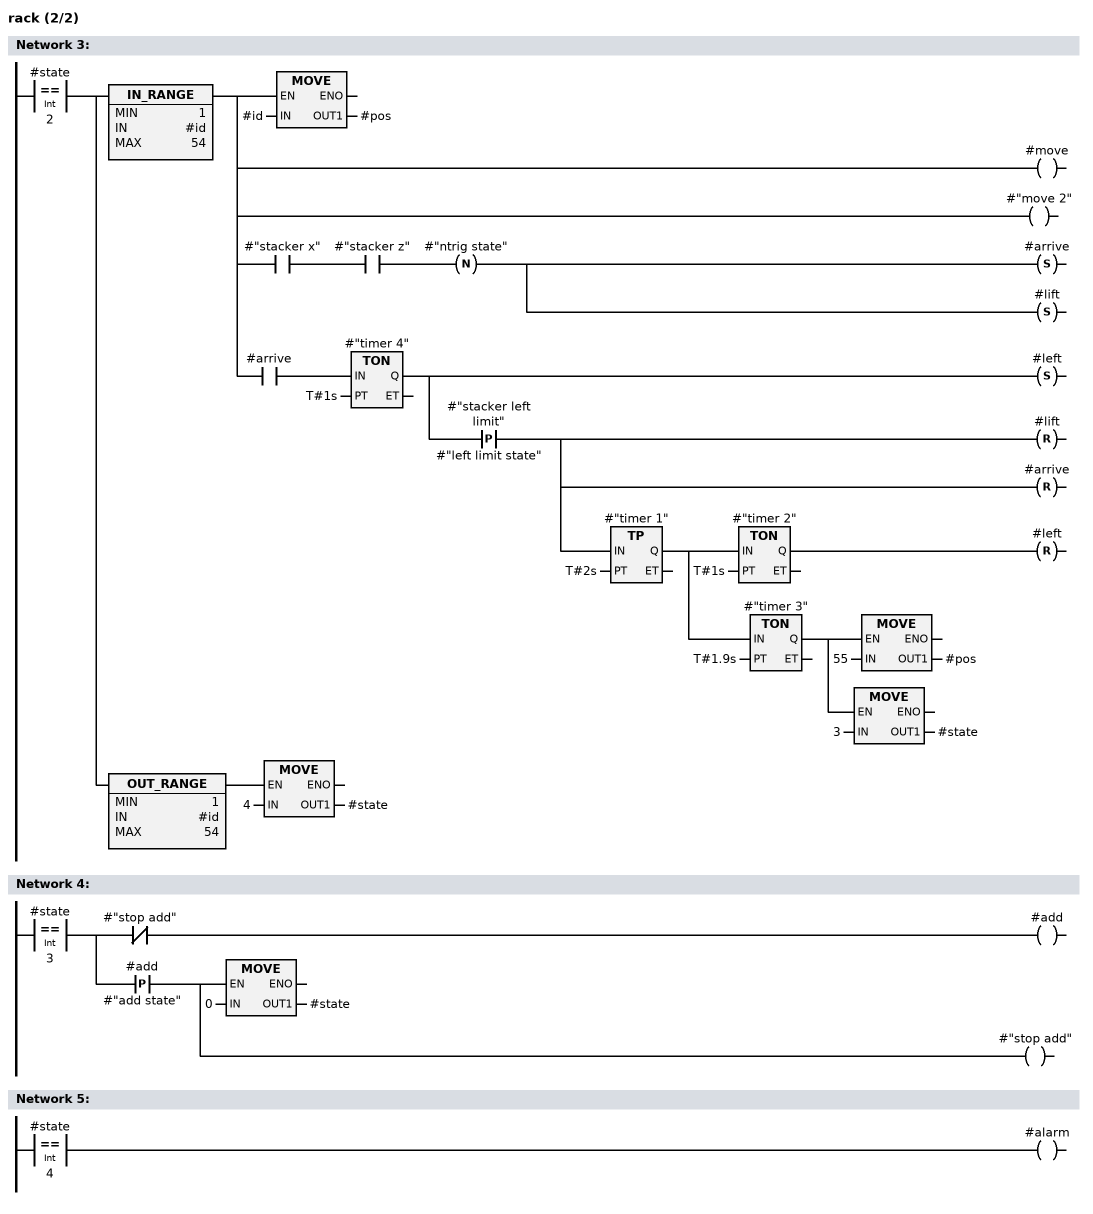
   #_w1 := #state = 2;
   #_w2 := #_w1 AND (1 <= #id) AND (#id <= 54);
   IF #_w2 THEN #pos := #id; END_IF;
   #move := #_w2;
   #"move 2" := #_w2;
   #_w3 := #_w2 AND #"stacker x" AND #"stacker z";
   #_w4 := NOT #_w3 AND #"ntrig state";   // falling edge
   #"ntrig state" := #_w3;
   IF #_w4 THEN
       #arrive := TRUE;
       #lift := TRUE;
   END_IF;
   #"timer 4".TON(IN := #_w2 AND #arrive, PT := T#1s);
   IF #"timer 4".Q THEN #left := TRUE; END_IF;
   #_w5 := #"timer 4".Q AND #"stacker left limit" AND NOT #"left limit state";   // rising edge of #"stacker left limit"
   #"left limit state" := #"stacker left limit";
   IF #_w5 THEN
       #lift := FALSE;
       #arrive := FALSE;
   END_IF;
   #"timer 1".TP(IN := #_w5, PT := T#2s);
   #"timer 2".TON(IN := #"timer 1".Q, PT := T#1s);
   IF #"timer 2".Q THEN #left := FALSE; END_IF;
   #"timer 3".TON(IN := #"timer 1".Q, PT := T#1.9s);
   IF #"timer 3".Q THEN
       #pos := 55;
       #state := 3;
   END_IF;
   IF #_w1 AND ((#id < 1) OR (#id > 54)) THEN #state := 4; END_IF;
END_REGION

REGION Network 4
   RUNG wire#powerrail
      { S7_Templates := "SrcType := Int" } EQ_Contact(in1 := #state, in2 := 3)
      wire#w1
      I_Contact( #"stop add" )
      Coil( #add )
   END_RUNG
   RUNG wire#w1
      P_Contact(operand := #add, bit := #"add state")
      wire#w2
      Move(in := 0, out1 => #state)
   END_RUNG
   RUNG wire#w2
      Coil( #"stop add" )
   END_RUNG
   // the same network as SCL:
   #_w1 := #state = 3;
   #add := #_w1 AND NOT #"stop add";
   #_w2 := #_w1 AND #add AND NOT #"add state";   // rising edge of #add
   #"add state" := #add;
   IF #_w2 THEN #state := 0; END_IF;
   #"stop add" := #_w2;
END_REGION

REGION Network 5
   RUNG wire#powerrail
      { S7_Templates := "SrcType := Int" } EQ_Contact(in1 := #state, in2 := 4)
      Coil( #alarm )
   END_RUNG
   // the same network as SCL:
   #alarm := #state = 4;
END_REGION
END_FUNCTION_BLOCK

FUNCTION "MHJ-PLC-Lab-Function-S71200" : Void   // FC9000, SCL
{ S7_Optimized_Access := 'TRUE' }
VERSION : 0.1
   VAR_TEMP
      rdTimeReturn : Int;
      outputTime : DTL;
      SyncVal : Byte;
      forVal : Int;
      forVal_2 : Int;
      Value : Byte;
   END_VAR
   VAR CONSTANT
      CompVal : Byte := 16#34;
      Value_01 : Byte := 16#11;
      Value_01_DW : DWord := 16#A165_D992;
      Value_02_DW : DWord := 16#58BE_4401;
   END_VAR
BEGIN

   #Value:=PEEK(area := 16#82,
        dbNumber := 0,
        byteOffset := 511);
   #Value := #Value + 1;

   POKE(area := 16#82,
        dbNumber := 0,
        byteOffset := 511,
        value := #Value);

   POKE(area:=16#81,
        dbNumber:=0,
        byteOffset:=1016,
        value:=#Value_01_DW);
   POKE(area := 16#81,
        dbNumber := 0,
        byteOffset := 1020,
        value := #Value_02_DW);

   POKE(area := 16#81,
        dbNumber := 0,
        byteOffset := 511,
        value := B#16#00);

   FOR #forVal := 0 TO 120 DO
       FOR #forVal_2:=0 TO 10 DO
           #rdTimeReturn:=RD_SYS_T(#outputTime);
           #rdTimeReturn := WR_SYS_T(#outputTime);
           #rdTimeReturn := RD_SYS_T(#outputTime);
           #rdTimeReturn := WR_SYS_T(#outputTime);
       END_FOR;
       #SyncVal:= PEEK(area := 16#81,
                      dbNumber := 0,
                      byteOffset := 511);
       IF #SyncVal = #CompVal THEN
          GOTO M_1;
       END_IF;
   END_FOR;
   RETURN;

   M_1:
   POKE(area := 16#81,
        dbNumber := 0,
        byteOffset := 511,
        value := B#16#0);
END_FUNCTION

ORGANIZATION_BLOCK "Main original"   // OB1, LAD, ProgramCycle
TITLE = "Main Program Sweep (Cycle)"
{ S7_Optimized_Access := 'TRUE' }
VERSION : 0.1
   VAR_INPUT
      Initial_Call : Bool;   // Initial call of this OB
      Remanence : Bool;   // =True, if remanent data are available
   END_VAR
   VAR_TEMP   // added for the SCL form of the ladder/FBD networks
      _w1 : Bool;
      _w2 : Bool;
      _w3 : Bool;
   END_VAR
BEGIN

REGION Network 1
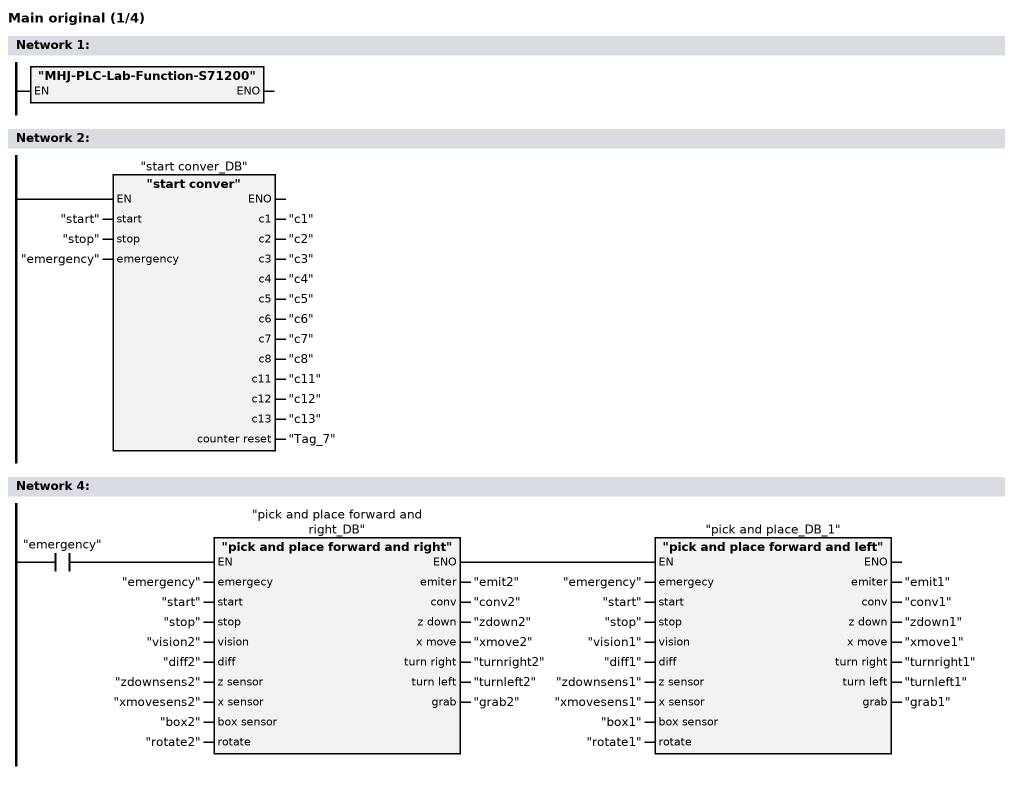
   RUNG wire#powerrail
      "MHJ-PLC-Lab-Function-S71200"()
   END_RUNG
   // the same network as SCL:
   "MHJ-PLC-Lab-Function-S71200"();
END_REGION

REGION Network 2
   RUNG wire#powerrail
      "start conver_DB"(start := "start", stop := "stop", emergency := "emergency", c1 => "c1", c2 => "c2", c3 => "c3", c4 => "c4", c5 => "c5", c6 => "c6", c7 => "c7", c8 => "c8", c11 => "c11", c12 => "c12", c13 => "c13", "counter reset" => "Tag_7")
   END_RUNG
   // the same network as SCL:
   "start conver_DB"(start := "start",   // "start conver"
                     stop := "stop",
                     emergency := "emergency",
                     c1 => "c1",
                     c2 => "c2",
                     c3 => "c3",
                     c4 => "c4",
                     c5 => "c5",
                     c6 => "c6",
                     c7 => "c7",
                     c8 => "c8",
                     c11 => "c11",
                     c12 => "c12",
                     c13 => "c13",
                     "counter reset" => "Tag_7");
END_REGION

REGION Network 4
   RUNG wire#powerrail
      Contact( "emergency" )
      "pick and place forward and right_DB"(emergecy := "emergency", start := "start", stop := "stop", vision := "vision2", diff := "diff2", "z sensor" := "zdownsens2", "x sensor" := "xmovesens2", "box sensor" := "box2", rotate := "rotate2", emiter => "emit2", conv => "conv2", "z down" => "zdown2", "x move" => "xmove2", "turn right" => "turnright2", "turn left" => "turnleft2", grab => "grab2")
      "pick and place_DB_1"(emergecy := "emergency", start := "start", stop := "stop", vision := "vision1", diff := "diff1", "z sensor" := "zdownsens1", "x sensor" := "xmovesens1", "box sensor" := "box1", rotate := "rotate1", emiter => "emit1", conv => "conv1", "z down" => "zdown1", "x move" => "xmove1", "turn right" => "turnright1", "turn left" => "turnleft1", grab => "grab1")
   END_RUNG
   // the same network as SCL:
   "pick and place forward and right_DB"(EN := "emergency",   // "pick and place forward and right"
                           emergecy := "emergency",
                           start := "start",
                           stop := "stop",
                           vision := "vision2",
                           diff := "diff2",
                           "z sensor" := "zdownsens2",
                           "x sensor" := "xmovesens2",
                           "box sensor" := "box2",
                           rotate := "rotate2",
                           emiter => "emit2",
                           conv => "conv2",
                           "z down" => "zdown2",
                           "x move" => "xmove2",
                           "turn right" => "turnright2",
                           "turn left" => "turnleft2",
                           grab => "grab2",
                           ENO => #_w1);
   IF #_w1 THEN
       "pick and place_DB_1"(emergecy := "emergency",   // "pick and place forward and left"
                             start := "start",
                             stop := "stop",
                             vision := "vision1",
                             diff := "diff1",
                             "z sensor" := "zdownsens1",
                             "x sensor" := "xmovesens1",
                             "box sensor" := "box1",
                             rotate := "rotate1",
                             emiter => "emit1",
                             conv => "conv1",
                             "z down" => "zdown1",
                             "x move" => "xmove1",
                             "turn right" => "turnright1",
                             "turn left" => "turnleft1",
                             grab => "grab1");
   END_IF;
END_REGION

REGION Network 5
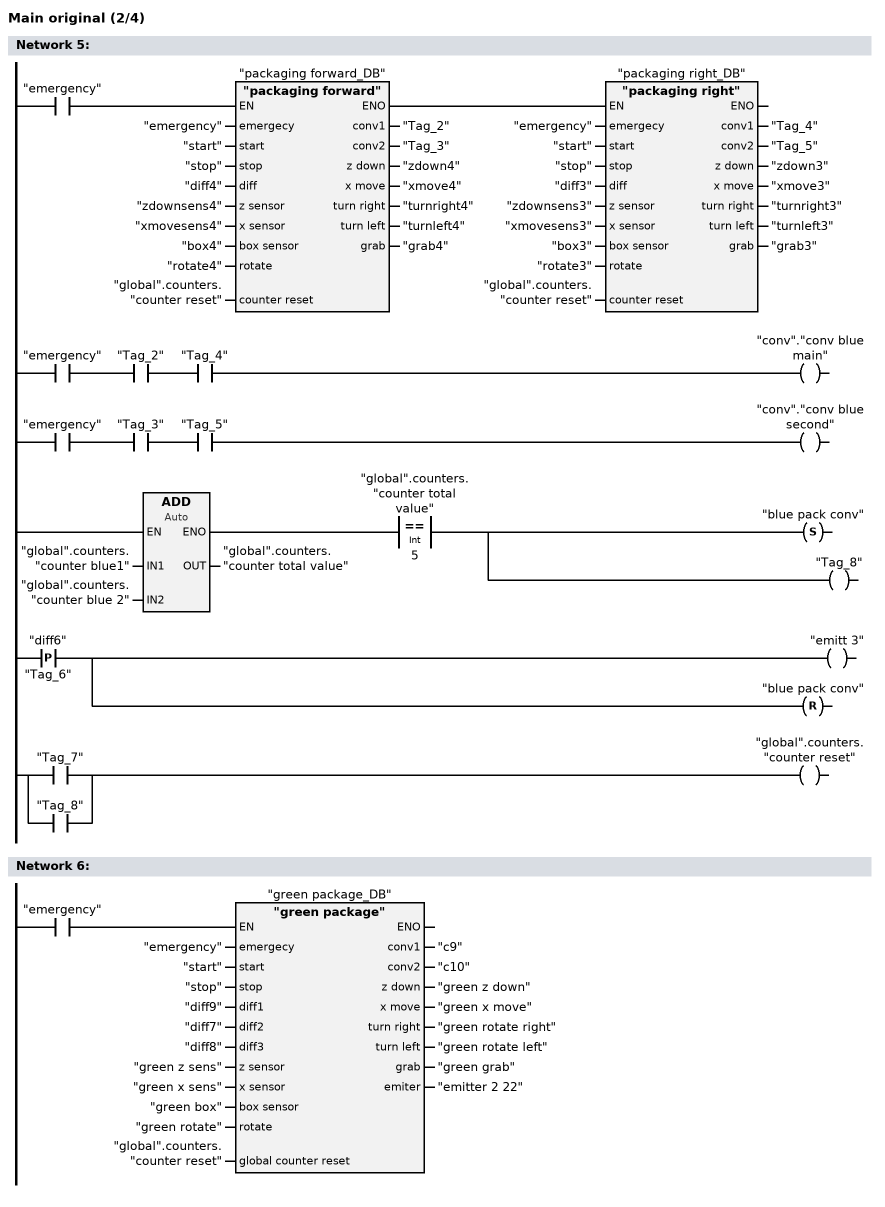
   RUNG wire#powerrail
      Contact( "emergency" )
      "packaging forward_DB"(emergecy := "emergency", start := "start", stop := "stop", diff := "diff4", "z sensor" := "zdownsens4", "x sensor" := "xmovesens4", "box sensor" := "box4", rotate := "rotate4", "counter reset" := "global".counters."counter reset", conv1 => "Tag_2", conv2 => "Tag_3", "z down" => "zdown4", "x move" => "xmove4", "turn right" => "turnright4", "turn left" => "turnleft4", grab => "grab4")
      "packaging right_DB"(emergecy := "emergency", start := "start", stop := "stop", diff := "diff3", "z sensor" := "zdownsens3", "x sensor" := "xmovesens3", "box sensor" := "box3", rotate := "rotate3", "counter reset" := "global".counters."counter reset", conv1 => "Tag_4", conv2 => "Tag_5", "z down" => "zdown3", "x move" => "xmove3", "turn right" => "turnright3", "turn left" => "turnleft3", grab => "grab3")
   END_RUNG
   RUNG wire#powerrail
      Contact( "emergency" )
      Contact( "Tag_2" )
      Contact( "Tag_4" )
      Coil( "conv"."conv blue main" )
   END_RUNG
   RUNG wire#powerrail
      Contact( "emergency" )
      Contact( "Tag_3" )
      Contact( "Tag_5" )
      Coil( "conv"."conv blue second" )
   END_RUNG
   RUNG wire#powerrail
      Add(in1 := "global".counters."counter blue1", in2 := "global".counters."counter blue 2", out => "global".counters."counter total value")
      { S7_Templates := "SrcType := Int" } EQ_Contact(in1 := "global".counters."counter total value", in2 := 5)
      wire#w1
      S_Coil( "blue pack conv" )
   END_RUNG
   RUNG wire#w1
      Coil( "Tag_8" )
   END_RUNG
   RUNG wire#powerrail
      P_Contact(operand := "diff6", bit := "Tag_6")
      wire#w2
      Coil( "emitt 3" )
   END_RUNG
   RUNG wire#w2
      R_Coil( "blue pack conv" )
   END_RUNG
   RUNG wire#powerrail
      Contact( "Tag_7" )
      wire#w3
      Coil( "global".counters."counter reset" )
   END_RUNG
   RUNG wire#powerrail
      Contact( "Tag_8" )
   END_RUNG wire#w3
   // the same network as SCL:
   "packaging forward_DB"(EN := "emergency",   // "packaging forward"
                          emergecy := "emergency",
                          start := "start",
                          stop := "stop",
                          diff := "diff4",
                          "z sensor" := "zdownsens4",
                          "x sensor" := "xmovesens4",
                          "box sensor" := "box4",
                          rotate := "rotate4",
                          "counter reset" := "global".counters."counter reset",
                          conv1 => "Tag_2",
                          conv2 => "Tag_3",
                          "z down" => "zdown4",
                          "x move" => "xmove4",
                          "turn right" => "turnright4",
                          "turn left" => "turnleft4",
                          grab => "grab4",
                          ENO => #_w1);
   IF #_w1 THEN
       "packaging right_DB"(emergecy := "emergency",   // "packaging right"
                            start := "start",
                            stop := "stop",
                            diff := "diff3",
                            "z sensor" := "zdownsens3",
                            "x sensor" := "xmovesens3",
                            "box sensor" := "box3",
                            rotate := "rotate3",
                            "counter reset" := "global".counters."counter reset",
                            conv1 => "Tag_4",
                            conv2 => "Tag_5",
                            "z down" => "zdown3",
                            "x move" => "xmove3",
                            "turn right" => "turnright3",
                            "turn left" => "turnleft3",
                            grab => "grab3");
   END_IF;
   "conv"."conv blue main" := "emergency" AND "Tag_2" AND "Tag_4";
   "conv"."conv blue second" := "emergency" AND "Tag_3" AND "Tag_5";
   "global".counters."counter total value" := "global".counters."counter blue1" + "global".counters."counter blue 2";
   #_w2 := "global".counters."counter total value" = 5;
   IF #_w2 THEN "blue pack conv" := TRUE; END_IF;
   "Tag_8" := #_w2;
   #_w3 := "diff6" AND NOT "Tag_6";   // rising edge of "diff6"
   "Tag_6" := "diff6";
   "emitt 3" := #_w3;
   IF #_w3 THEN "blue pack conv" := FALSE; END_IF;
   "global".counters."counter reset" := "Tag_7" OR "Tag_8";
END_REGION

REGION Network 6
   RUNG wire#powerrail
      Contact( "emergency" )
      "green package_DB"(emergecy := "emergency", start := "start", stop := "stop", diff1 := "diff9", diff2 := "diff7", diff3 := "diff8", "z sensor" := "green z sens", "x sensor" := "green x sens", "box sensor" := "green box", rotate := "green rotate", "global counter reset" := "global".counters."counter reset", conv1 => "c9", conv2 => "c10", "z down" => "green z down", "x move" => "green x move", "turn right" => "green rotate right", "turn left" => "green rotate left", grab => "green grab", emiter => "emitter 2 22")
   END_RUNG
   // the same network as SCL:
   IF "emergency" THEN
       "green package_DB"(emergecy := "emergency",   // "green package"
                          start := "start",
                          stop := "stop",
                          diff1 := "diff9",
                          diff2 := "diff7",
                          diff3 := "diff8",
                          "z sensor" := "green z sens",
                          "x sensor" := "green x sens",
                          "box sensor" := "green box",
                          rotate := "green rotate",
                          "global counter reset" := "global".counters."counter reset",
                          conv1 => "c9",
                          conv2 => "c10",
                          "z down" => "green z down",
                          "x move" => "green x move",
                          "turn right" => "green rotate right",
                          "turn left" => "green rotate left",
                          grab => "green grab",
                          emiter => "emitter 2 22");
   END_IF;
END_REGION

REGION Network 8
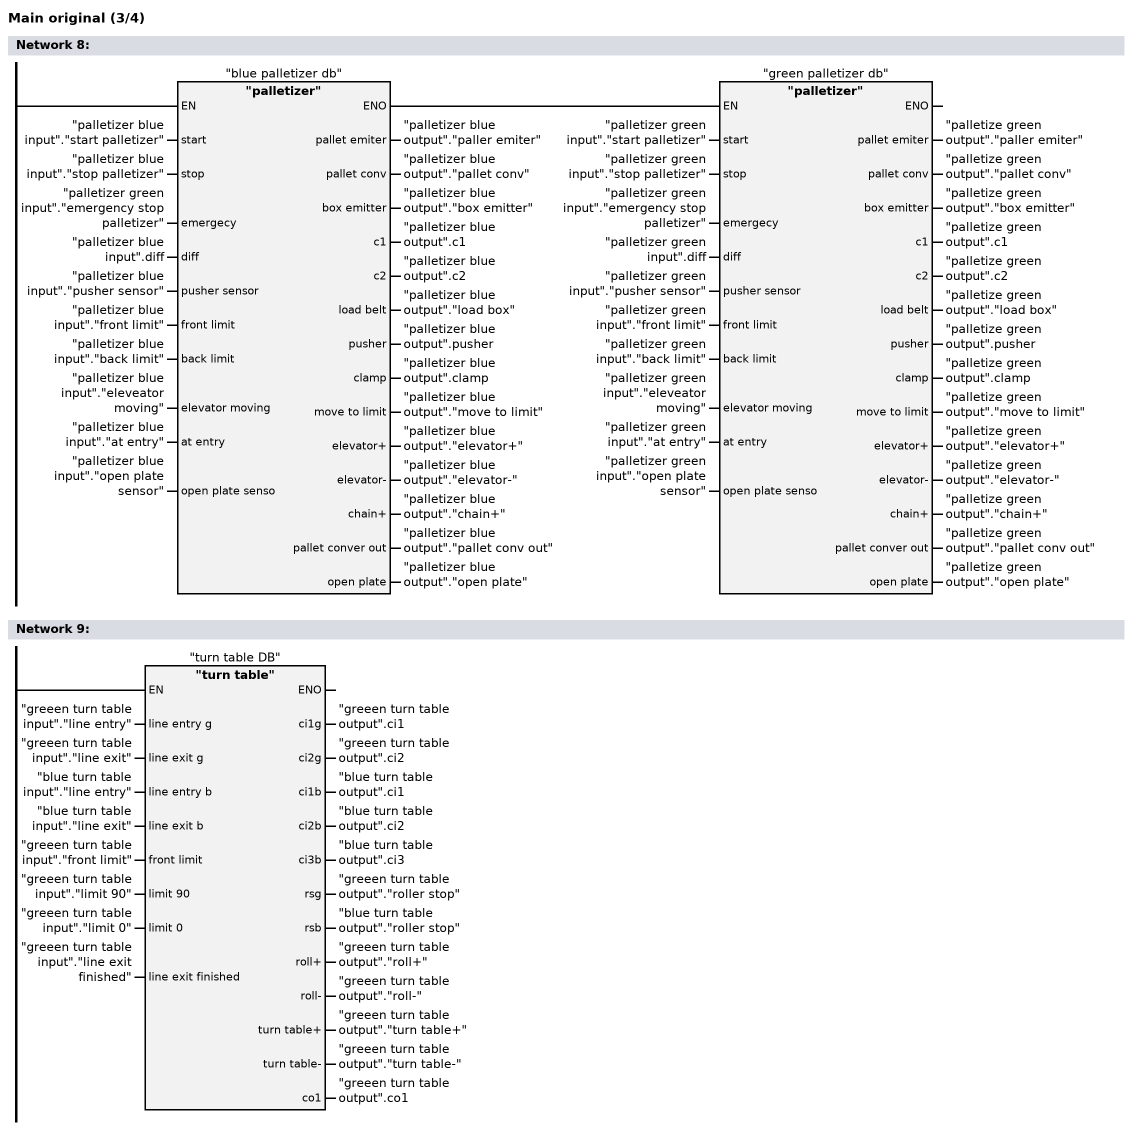
   RUNG wire#powerrail
      "blue palletizer db"(start := "palletizer blue input"."start palletizer", stop := "palletizer blue input"."stop palletizer", emergecy := "palletizer green input"."emergency stop palletizer", diff := "palletizer blue input".diff, "pusher sensor" := "palletizer blue input"."pusher sensor", "front limit" := "palletizer blue input"."front limit", "back limit" := "palletizer blue input"."back limit", "elevator moving" := "palletizer blue input"."eleveator moving", "at entry" := "palletizer blue input"."at entry", "open plate senso" := "palletizer blue input"."open plate sensor", "pallet emiter" => "palletizer blue output"."paller emiter", "pallet conv" => "palletizer blue output"."pallet conv", "box emitter" => "palletizer blue output"."box emitter", c1 => "palletizer blue output".c1, c2 => "palletizer blue output".c2, "load belt" => "palletizer blue output"."load box", pusher => "palletizer blue output".pusher, clamp => "palletizer blue output".clamp, "move to limit" => "palletizer blue output"."move to limit", "elevator+" => "palletizer blue output"."elevator+", "elevator-" => "palletizer blue output"."elevator-", "chain+" => "palletizer blue output"."chain+", "pallet conver out" => "palletizer blue output"."pallet conv out", "open plate" => "palletizer blue output"."open plate")
      "green palletizer db"(start := "palletizer green input"."start palletizer", stop := "palletizer green input"."stop palletizer", emergecy := "palletizer green input"."emergency stop palletizer", diff := "palletizer green input".diff, "pusher sensor" := "palletizer green input"."pusher sensor", "front limit" := "palletizer green input"."front limit", "back limit" := "palletizer green input"."back limit", "elevator moving" := "palletizer green input"."eleveator moving", "at entry" := "palletizer green input"."at entry", "open plate senso" := "palletizer green input"."open plate sensor", "pallet emiter" => "palletize green output"."paller emiter", "pallet conv" => "palletize green output"."pallet conv", "box emitter" => "palletize green output"."box emitter", c1 => "palletize green output".c1, c2 => "palletize green output".c2, "load belt" => "palletize green output"."load box", pusher => "palletize green output".pusher, clamp => "palletize green output".clamp, "move to limit" => "palletize green output"."move to limit", "elevator+" => "palletize green output"."elevator+", "elevator-" => "palletize green output"."elevator-", "chain+" => "palletize green output"."chain+", "pallet conver out" => "palletize green output"."pallet conv out", "open plate" => "palletize green output"."open plate")
   END_RUNG
   // the same network as SCL:
   "blue palletizer db"(start := "palletizer blue input"."start palletizer",   // "palletizer"
                        stop := "palletizer blue input"."stop palletizer",
                        emergecy := "palletizer green input"."emergency stop palletizer",
                        diff := "palletizer blue input".diff,
                        "pusher sensor" := "palletizer blue input"."pusher sensor",
                        "front limit" := "palletizer blue input"."front limit",
                        "back limit" := "palletizer blue input"."back limit",
                        "elevator moving" := "palletizer blue input"."eleveator moving",
                        "at entry" := "palletizer blue input"."at entry",
                        "open plate senso" := "palletizer blue input"."open plate sensor",
                        "pallet emiter" => "palletizer blue output"."paller emiter",
                        "pallet conv" => "palletizer blue output"."pallet conv",
                        "box emitter" => "palletizer blue output"."box emitter",
                        c1 => "palletizer blue output".c1,
                        c2 => "palletizer blue output".c2,
                        "load belt" => "palletizer blue output"."load box",
                        pusher => "palletizer blue output".pusher,
                        clamp => "palletizer blue output".clamp,
                        "move to limit" => "palletizer blue output"."move to limit",
                        "elevator+" => "palletizer blue output"."elevator+",
                        "elevator-" => "palletizer blue output"."elevator-",
                        "chain+" => "palletizer blue output"."chain+",
                        "pallet conver out" => "palletizer blue output"."pallet conv out",
                        "open plate" => "palletizer blue output"."open plate",
                        ENO => #_w1);
   IF #_w1 THEN
       "green palletizer db"(start := "palletizer green input"."start palletizer",   // "palletizer"
                             stop := "palletizer green input"."stop palletizer",
                             emergecy := "palletizer green input"."emergency stop palletizer",
                             diff := "palletizer green input".diff,
                             "pusher sensor" := "palletizer green input"."pusher sensor",
                             "front limit" := "palletizer green input"."front limit",
                             "back limit" := "palletizer green input"."back limit",
                             "elevator moving" := "palletizer green input"."eleveator moving",
                             "at entry" := "palletizer green input"."at entry",
                             "open plate senso" := "palletizer green input"."open plate sensor",
                             "pallet emiter" => "palletize green output"."paller emiter",
                             "pallet conv" => "palletize green output"."pallet conv",
                             "box emitter" => "palletize green output"."box emitter",
                             c1 => "palletize green output".c1,
                             c2 => "palletize green output".c2,
                             "load belt" => "palletize green output"."load box",
                             pusher => "palletize green output".pusher,
                             clamp => "palletize green output".clamp,
                             "move to limit" => "palletize green output"."move to limit",
                             "elevator+" => "palletize green output"."elevator+",
                             "elevator-" => "palletize green output"."elevator-",
                             "chain+" => "palletize green output"."chain+",
                             "pallet conver out" => "palletize green output"."pallet conv out",
                             "open plate" => "palletize green output"."open plate");
   END_IF;
END_REGION

REGION Network 9
   RUNG wire#powerrail
      "turn table DB"("line entry g" := "greeen turn table input"."line entry", "line exit g" := "greeen turn table input"."line exit", "line entry b" := "blue turn table input"."line entry", "line exit b" := "blue turn table input"."line exit", "front limit" := "greeen turn table input"."front limit", "limit 90" := "greeen turn table input"."limit 90", "limit 0" := "greeen turn table input"."limit 0", "line exit finished" := "greeen turn table input"."line exit finished", ci1g => "greeen turn table output".ci1, ci2g => "greeen turn table output".ci2, ci1b => "blue turn table output".ci1, ci2b => "blue turn table output".ci2, ci3b => "blue turn table output".ci3, rsg => "greeen turn table output"."roller stop", rsb => "blue turn table output"."roller stop", "roll+" => "greeen turn table output"."roll+", "roll-" => "greeen turn table output"."roll-", "turn table+" => "greeen turn table output"."turn table+", "turn table-" => "greeen turn table output"."turn table-", co1 => "greeen turn table output".co1)
   END_RUNG
   // the same network as SCL:
   "turn table DB"("line entry g" := "greeen turn table input"."line entry",   // "turn table"
                   "line exit g" := "greeen turn table input"."line exit",
                   "line entry b" := "blue turn table input"."line entry",
                   "line exit b" := "blue turn table input"."line exit",
                   "front limit" := "greeen turn table input"."front limit",
                   "limit 90" := "greeen turn table input"."limit 90",
                   "limit 0" := "greeen turn table input"."limit 0",
                   "line exit finished" := "greeen turn table input"."line exit finished",
                   ci1g => "greeen turn table output".ci1,
                   ci2g => "greeen turn table output".ci2,
                   ci1b => "blue turn table output".ci1,
                   ci2b => "blue turn table output".ci2,
                   ci3b => "blue turn table output".ci3,
                   rsg => "greeen turn table output"."roller stop",
                   rsb => "blue turn table output"."roller stop",
                   "roll+" => "greeen turn table output"."roll+",
                   "roll-" => "greeen turn table output"."roll-",
                   "turn table+" => "greeen turn table output"."turn table+",
                   "turn table-" => "greeen turn table output"."turn table-",
                   co1 => "greeen turn table output".co1);
END_REGION

REGION Network 10
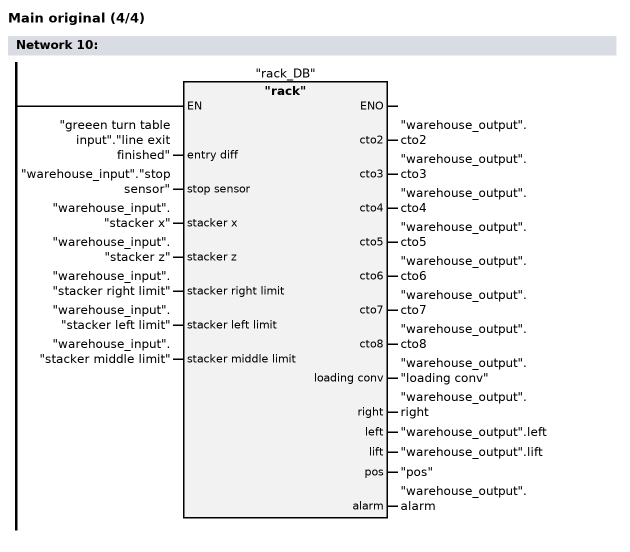
   RUNG wire#powerrail
      "rack_DB"("entry diff" := "greeen turn table input"."line exit finished", "stop sensor" := "warehouse_input"."stop sensor", "stacker x" := "warehouse_input"."stacker x", "stacker z" := "warehouse_input"."stacker z", "stacker right limit" := "warehouse_input"."stacker right limit", "stacker left limit" := "warehouse_input"."stacker left limit", "stacker middle limit" := "warehouse_input"."stacker middle limit", cto2 => "warehouse_output".cto2, cto3 => "warehouse_output".cto3, cto4 => "warehouse_output".cto4, cto5 => "warehouse_output".cto5, cto6 => "warehouse_output".cto6, cto7 => "warehouse_output".cto7, cto8 => "warehouse_output".cto8, "loading conv" => "warehouse_output"."loading conv", right => "warehouse_output".right, left => "warehouse_output".left, lift => "warehouse_output".lift, pos => "pos", alarm => "warehouse_output".alarm)
   END_RUNG
   // the same network as SCL:
   "rack_DB"("entry diff" := "greeen turn table input"."line exit finished",   // "rack"
             "stop sensor" := "warehouse_input"."stop sensor",
             "stacker x" := "warehouse_input"."stacker x",
             "stacker z" := "warehouse_input"."stacker z",
             "stacker right limit" := "warehouse_input"."stacker right limit",
             "stacker left limit" := "warehouse_input"."stacker left limit",
             "stacker middle limit" := "warehouse_input"."stacker middle limit",
             cto2 => "warehouse_output".cto2,
             cto3 => "warehouse_output".cto3,
             cto4 => "warehouse_output".cto4,
             cto5 => "warehouse_output".cto5,
             cto6 => "warehouse_output".cto6,
             cto7 => "warehouse_output".cto7,
             cto8 => "warehouse_output".cto8,
             "loading conv" => "warehouse_output"."loading conv",
             right => "warehouse_output".right,
             left => "warehouse_output".left,
             lift => "warehouse_output".lift,
             pos => "pos",
             alarm => "warehouse_output".alarm);
END_REGION
END_ORGANIZATION_BLOCK